// TwinCAT 3 PLC project PLCMotionOOP
// ProgramVersion: 3.1.4024.0
// libraries:
//   Tc2_MC2, * (Beckhoff Automation GmbH)
//   Tc2_Standard, * (Beckhoff Automation GmbH)
//   Tc2_System, * (Beckhoff Automation GmbH)
//   Tc3_Module, * (Beckhoff Automation GmbH)
// project tree:
//   MotionOOP/PLCOpenDefination/BeckhoffImplementation/ Axis.TcPOU
//   MotionOOP/PLCOpenDefination/Part1Definition/Enums/ AXIS_DIRECTION.TcDUT, AXIS_STATUS.TcDUT, MC_BUFFER_MODE.TcDUT, MC_COMBINE_MODE.TcDUT, MC_Direction.TcDUT, MC_Error.TcDUT, MC_ExecutionMode.TcDUT, MC_Source.TcDUT, MC_StartMode.TcDUT, MC_SYNC_MODE.TcDUT, MOTION_STATUS.TcDUT
//   MotionOOP/PLCOpenDefination/Part1Definition/GlobalConstants/ Constants.TcGVL
//   MotionOOP/PLCOpenDefination/Part1Definition/Interfaces/ itfAxis.TcIO, itfAxisCommand.TcIO, itfCamTable.TcIO, itfCommand.TcIO, itfContinuousAxisCommand.TcIO, itfSynchronizedAxisCommand.TcIO
//   MotionOOP/PLCOpenDefination/Part1Definition/Structs/ MC_CAM_REF.TcDUT, MC_COMMAND_REF.TcDUT
//   / PlcTask.TcTTO
//   POUs/ MAIN.TcPOU
// real-time tasks:
//   TASK PlcTask: cycle T#10ms, priority 20, ADS port 350
//   TASK PlcTask1: cycle T#10ms, priority 21, ADS port 351

CONFIGURATION PLCMotionOOP
    RESOURCE PLC ON TwinCAT3
        TASK PlcTask(INTERVAL := T#10ms, PRIORITY := 21);
        PROGRAM MAIN WITH PlcTask : MAIN;
    END_RESOURCE
END_CONFIGURATION

// ---- MotionOOP/PLCOpenDefination/Part1Definition/Enums/AXIS_DIRECTION.TcDUT
{attribute 'qualified_only' := ''}
{attribute 'strict' := ''}
TYPE AXIS_DIRECTION :
(
	DirectionPositive := 0,
	DirectionNegative := 1
);
END_TYPE

// ---- MotionOOP/PLCOpenDefination/Part1Definition/Enums/AXIS_STATUS.TcDUT
{attribute 'qualified_only' := ''}
{attribute 'strict' := ''}
TYPE AXIS_STATUS :
(
	ErrorStop := 0,
	Disabled := 1,
	Stopping := 2,
	Homing := 3,
	Standstill := 4,
	DiscreteMotion := 5,
	ContinuousMotion := 6,
	SynchronizedMotion := 7
);
END_TYPE

// ---- MotionOOP/PLCOpenDefination/Part1Definition/Enums/MC_BUFFER_MODE.TcDUT
{attribute 'qualified_only' := ''}
{attribute 'strict' := ''}
TYPE MC_BUFFER_MODE :
(
	mcAborting := 0,
	mcBuffered := 1,
	mcBlendingLow := 2,
	mcBlendingPrevious := 3,
	mcBlendingNext := 4,
	mcBlendingHigh := 5
);
END_TYPE

// ---- MotionOOP/PLCOpenDefination/Part1Definition/Enums/MC_COMBINE_MODE.TcDUT
{attribute 'qualified_only' := ''}
{attribute 'strict' := ''}
TYPE MC_COMBINE_MODE :
(
	enum_member := 0
);
END_TYPE

// ---- MotionOOP/PLCOpenDefination/Part1Definition/Enums/MC_Direction.TcDUT
{attribute 'qualified_only' := ''}
{attribute 'strict' := ''}
TYPE MC_Direction :
(
	mcPositiveDirection := 0,
	mcShortestWay := 1,
	mcNegativeDirection := 2,
	mcCurrentDirection := 3
);
END_TYPE

// ---- MotionOOP/PLCOpenDefination/Part1Definition/Enums/MC_Error.TcDUT
///{attribute 'conditionalshow' := 'SomeText'}
///{attribute 'conditionalshow'}
///{attribute 'hide'}
{attribute 'qualified_only' := ''}
TYPE MC_Error :
(
	NO_ERROR,
	TIME_OUT
);
END_TYPE

// ---- MotionOOP/PLCOpenDefination/Part1Definition/Enums/MC_ExecutionMode.TcDUT
{attribute 'qualified_only' := ''}
{attribute 'strict' := ''}
TYPE MC_ExecutionMode :
(
	mcImmediatly := 0,
	mcQueue := 1
);
END_TYPE

// ---- MotionOOP/PLCOpenDefination/Part1Definition/Enums/MC_Source.TcDUT
{attribute 'qualified_only' := ''}
{attribute 'strict' := ''}
TYPE MC_Source :
(
	mcSetValue := 0,
	mcActualValue := 1
);
END_TYPE

// ---- MotionOOP/PLCOpenDefination/Part1Definition/Enums/MC_StartMode.TcDUT
{attribute 'qualified_only' := ''}
{attribute 'strict' := ''}
TYPE MC_StartMode :
(
	mcAbsolute := 0,
	mcRelative := 1,
	mcRampIn := 2
);
END_TYPE

// ---- MotionOOP/PLCOpenDefination/Part1Definition/Enums/MC_SYNC_MODE.TcDUT
{attribute 'qualified_only' := ''}
{attribute 'strict' := ''}
TYPE MC_SYNC_MODE :
(
	enum_member := 0
);
END_TYPE

// ---- MotionOOP/PLCOpenDefination/Part1Definition/Enums/MOTION_STATUS.TcDUT
{attribute 'qualified_only' := ''}
{attribute 'strict' := ''}
TYPE MOTION_STATUS :
(
	ConstantVelocity := 0,
	Accelerating := 1,
	Decelerating := 2
);
END_TYPE

// ---- MotionOOP/PLCOpenDefination/Part1Definition/Structs/MC_CAM_REF.TcDUT
TYPE MC_CAM_REF :
STRUCT
END_STRUCT
END_TYPE

// ---- MotionOOP/PLCOpenDefination/Part1Definition/Structs/MC_COMMAND_REF.TcDUT
TYPE MC_COMMAND_REF :
STRUCT
	CommandId: INT;
END_STRUCT
END_TYPE

// ---- MotionOOP/PLCOpenDefination/Part1Definition/GlobalConstants/Constants.TcGVL
///{attribute 'conditionalshow' := 'SomeText'}
///{attribute 'conditionalshow'}
///{attribute 'hide'}
VAR_GLOBAL
END_VAR

// ---- MotionOOP/PLCOpenDefination/Part1Definition/Interfaces/itfAxis.TcIO
INTERFACE itfAxis

METHOD AccelerationProfile : itfCommand
VAR_INPUT
	TimeScale: REAL;
	AccelerationScale: REAL;
	Offset: REAL;
	BufferMode: MC_BUFFER_MODE;
END_VAR
END_METHOD

PROPERTY ActualPosition : REAL
GET
END_GET
END_PROPERTY

PROPERTY ActualTorque : REAL
GET
END_GET
END_PROPERTY

PROPERTY ActualVelocity : REAL
GET
END_GET
END_PROPERTY

PROPERTY AxisWarning : BOOL
GET
END_GET
END_PROPERTY

METHOD CamIn : itfSynchronizedAxisCommand
VAR_INPUT
	Master: itfAxis;
	MasterOffset: REAL;
	SlaveOffset: REAL;
	MasterScaling: REAL;
	SlaveScaling: REAL;
	MasterStartDistance: REAL;
	MasterSyncPosition: REAL;
	StartMode: MC_StartMode;
	MasterValueSource: MC_Source;
	CamTable: itfCamTable;
	BufferMode: MC_BUFFER_MODE;
END_VAR
END_METHOD

METHOD CombineAxes : itfSynchronizedAxisCommand
VAR_INPUT
	Master1: itfAxis;
	Master2: itfAxis;
	CombineMode: MC_COMBINE_MODE;
	GearRatioNumeratorM1: INT;
	GearRatioDenominatorM1: INT;
	GearRatioNumeratorM2: INT;
	GearRatioDenominatorM2: INT;
	MasterValueSourceM1: MC_SOURCE;
	MasterValueSourceM2: MC_SOURCE;
	BufferMode: MC_BUFFER_MODE;
END_VAR
END_METHOD

PROPERTY CommunicationReady : BOOL
GET
END_GET
END_PROPERTY

PROPERTY Direction : AXIS_DIRECTION
GET
END_GET
END_PROPERTY

PROPERTY ErrorId : WORD
GET
END_GET
END_PROPERTY

METHOD GearIn : itfSynchronizedAxisCommand
VAR_INPUT
	Master: itfAxis;
	Ratio: REAL;
	MasterValueSource: INT;
	Acceleration: REAL;
	Deceleration: REAL;
	Jerk: REAL;
	BufferMode: MC_BUFFER_MODE;
END_VAR
END_METHOD

METHOD GearInPos : itfSynchronizedAxisCommand
VAR_INPUT
	Master: itfAxis;
	RatioNumerator: REAL;
	RatioDenominator: REAL;
	MasterValueSource: MC_SOURCE;
	MasterSyncPosition: REAL;
	SlaveSyncPosition: REAL;
	SyncMode: MC_SYNC_MODE;
	MasterStartDistance: REAL;
	Velocity: REAL;
	Acceleration: REAL;
	Deceleration: REAL;
	Jerk: REAL;
	BufferMode: MC_BUFFER_MODE;
END_VAR
END_METHOD

METHOD Halt : itfAxisCommand
VAR_INPUT
	Deceleration: REAL;
	Jerk: REAL;
	BufferMode: MC_BUFFER_MODE;
END_VAR
END_METHOD

METHOD HaltSuperimposed : itfAxisCommand
VAR_INPUT
	Deceleration: REAL;
	Jerk: REAL;
END_VAR
END_METHOD

METHOD Home : itfAxisCommand
VAR_INPUT
	Position: REAL;
	Velocity: REAL;
	EndVelocity: REAL;
	Acceleration: REAL;
	Deceleration: REAL;
	Jerk: REAL;
	Direction: MC_Direction;
	HomingMode: INT;
	BufferMode: MC_BUFFER_MODE;
END_VAR
END_METHOD

PROPERTY HomeAbsSwitch : BOOL
GET
END_GET
END_PROPERTY

PROPERTY IsHomed : BOOL
GET
END_GET
END_PROPERTY

PROPERTY LimitSwitchNegative : BOOL
GET
END_GET
END_PROPERTY

PROPERTY LimitSwitchPositive : BOOL
GET
END_GET
END_PROPERTY

PROPERTY MotionStatus : MOTION_STATUS
GET
END_GET
END_PROPERTY

METHOD MoveAbsolute : itfAxisCommand
VAR_INPUT
	Position: REAL;
	Velocity: REAL;
	Acceleration: REAL;
	Deceleration: REAL;
	Jerk: REAL;
	Direction: MC_Direction;
	BufferMode: MC_BUFFER_MODE;
END_VAR
END_METHOD

METHOD MoveAdditive : itfAxisCommand
VAR_INPUT
	Distance: REAL;
	Velocity: REAL;
	Acceleration: REAL;
	Deceleration: REAL;
	Jerk: REAL;
	BufferMode: MC_BUFFER_MODE;
END_VAR
END_METHOD

METHOD MoveContinuousAbsolute : itfContinuousAxisCommand
VAR_INPUT
	Position: REAL;
	EndVelocity: REAL;
	Velocity: REAL;
	Acceleration: REAL;
	Deceleration: REAL;
	Jerk: REAL;
	Direction: MC_DIRECTION;
	BufferMode: MC_BUFFER_MODE;
END_VAR
END_METHOD

METHOD MoveContinuousRelative : itfContinuousAxisCommand
VAR_INPUT
	Distance: REAL;
	EndVelocity: REAL;
	Velocity: REAL;
	Acceleration: REAL;
	Deceleration: REAL;
	Jerk: REAL;
	Direction: MC_DIRECTION;
	BufferMode: MC_BUFFER_MODE;
END_VAR
END_METHOD

METHOD MoveRelative : itfAxisCommand
VAR_INPUT
	Distance: REAL;
	Velocity: REAL;
	Acceleration: REAL;
	Deceleration: REAL;
	Jerk: REAL;
	BufferMode: MC_BUFFER_MODE;
END_VAR
END_METHOD

METHOD MoveSuperimposed : itfAxisCommand
VAR_INPUT
	Distance: REAL;
	VelocityDiff: REAL;
	Acceleration: REAL;
	Deceleration: REAL;
	Jerk: REAL;
END_VAR
END_METHOD

METHOD MoveVelocity : itfContinuousAxisCommand
VAR_INPUT
	Velocity: REAL;
	Acceleration: REAL;
	Deceleration: REAL;
	Jerk: REAL;
	Direction: MC_Direction;
	BufferMode: MC_BUFFER_MODE;
END_VAR
END_METHOD

METHOD PhasingAbsolute : itfSynchronizedAxisCommand
VAR_INPUT
	Master: itfAxis;
	PhaseShift: REAL;
	Velocity: REAL;
	Acceleration: REAL;
	Deceleration: REAL;
	Jerk: REAL;
	BufferMode: MC_BUFFER_MODE;
END_VAR
END_METHOD

METHOD PhasingRelative : itfSynchronizedAxisCommand
VAR_INPUT
	Master: itfAxis;
	PhaseShift: REAL;
	Velocity: REAL;
	Acceleration: REAL;
	Deceleration: REAL;
	Jerk: REAL;
	BufferMode: MC_BUFFER_MODE;
END_VAR
END_METHOD

METHOD PositionProfile : itfCommand
VAR_INPUT
	TimeScale: REAL;
	PositionScale: REAL;
	Offset: REAL;
	BufferMode: MC_BUFFER_MODE;
END_VAR
END_METHOD

METHOD Power : itfCommand
VAR_INPUT
	Enable: BOOL;
	EnablePositive: BOOL;
	EnableNegative: BOOL;
END_VAR
END_METHOD

PROPERTY PowerOn : BOOL
GET
END_GET
END_PROPERTY

METHOD ReadBoolParameter : MC_Error
VAR_INPUT
	ParameterNumber: INT;
END_VAR
VAR_OUTPUT
	Value: BOOL;
END_VAR
END_METHOD

METHOD ReadParameter : MC_Error
VAR_INPUT
	ParameterNumber: INT;
END_VAR
VAR_OUTPUT
	Value: REAL;
END_VAR
END_METHOD

PROPERTY ReadyForPowerOn : BOOL
GET
END_GET
END_PROPERTY

METHOD Release : MC_Error
END_METHOD

METHOD Reset : itfCommand
END_METHOD

METHOD SetOverride : MC_Error
VAR_INPUT
	VelFactor: REAL;
	AccFactor: REAL;
	JerkFactor: REAL;
END_VAR
END_METHOD

METHOD SetPosition : itfCommand
VAR_INPUT
	Position: REAL;
	Relative: BOOL;
	ExecutionMode: MC_ExecutionMode;
END_VAR
END_METHOD

PROPERTY Simulation : BOOL
GET
END_GET
END_PROPERTY

PROPERTY Status : AXIS_STATUS
GET
END_GET
END_PROPERTY

METHOD Stop : itfAxisCommand
VAR_INPUT
	Deceleration: REAL;
	Jerk: REAL;
END_VAR
END_METHOD

METHOD TorqueControl : itfAxisCommand
VAR_INPUT
	Torque: REAL;
	TorqueRamp: REAL;
	Velocity: REAL;
	Acceleration: REAL;
	Deceleration: REAL;
	Jerk: REAL;
	Direction: MC_DIRECTION;
	BufferMode: MC_BUFFER_MODE;
END_VAR
END_METHOD

METHOD VelocityProfile : itfCommand
VAR_INPUT
	TimeScale: REAL;
	VelocityScale: REAL;
	Offset: REAL;
	BufferMode: MC_BUFFER_MODE;
END_VAR
END_METHOD

METHOD WriteBoolParameter : MC_Error
VAR_INPUT
	ParameterNumber: INT;
	Value: BOOL;
END_VAR
END_METHOD

METHOD WriteParameter : MC_Error
VAR_INPUT
	ParameterNumber: INT;
	Value: REAL;
END_VAR
END_METHOD

END_INTERFACE

// ---- MotionOOP/PLCOpenDefination/Part1Definition/Interfaces/itfAxisCommand.TcIO
INTERFACE itfAxisCommand EXTENDS itfCommand

METHOD Update : MC_Error
VAR_INPUT
	Position: REAL;
	Velocity: REAL;
	EndVelocity: REAL;
	Acceleration: REAL;
	Deceleration: REAL;
	Jerk: REAL;
END_VAR
END_METHOD

END_INTERFACE

// ---- MotionOOP/PLCOpenDefination/Part1Definition/Interfaces/itfCamTable.TcIO
INTERFACE itfCamTable

METHOD Select : itfCommand
VAR_INPUT
	Periodic: BOOL;
	MasterAbsolute: BOOL;
	SlaveAbsolute: BOOL;
	CamTable: MC_CAM_REF;
END_VAR
END_METHOD

END_INTERFACE

// ---- MotionOOP/PLCOpenDefination/Part1Definition/Interfaces/itfCommand.TcIO
INTERFACE itfCommand

METHOD Abort : MC_Error
END_METHOD

PROPERTY Active : BOOL
GET
END_GET
END_PROPERTY

PROPERTY Busy : BOOL
GET
END_GET
END_PROPERTY

PROPERTY Command : MC_COMMAND_REF
GET
END_GET
END_PROPERTY

PROPERTY CommandAborted : BOOL
GET
END_GET
END_PROPERTY

PROPERTY Done : BOOL
GET
END_GET
END_PROPERTY

PROPERTY Error : BOOL
GET
END_GET
END_PROPERTY

PROPERTY ErrorId : MC_Error
GET
END_GET
END_PROPERTY

METHOD Wait : MC_Error
VAR_INPUT
	Timeout: TIME;
	AbortOnTimeout: BOOL;
END_VAR
END_METHOD

END_INTERFACE

// ---- MotionOOP/PLCOpenDefination/Part1Definition/Interfaces/itfContinuousAxisCommand.TcIO
INTERFACE itfContinuousAxisCommand EXTENDS itfAxisCommand

PROPERTY InVelocity : BOOL
GET
END_GET
END_PROPERTY

END_INTERFACE

// ---- MotionOOP/PLCOpenDefination/Part1Definition/Interfaces/itfSynchronizedAxisCommand.TcIO
INTERFACE itfSynchronizedAxisCommand EXTENDS itfAxisCommand

PROPERTY InSync : BOOL
GET
END_GET
END_PROPERTY

END_INTERFACE

// ---- POUs/MAIN.TcPOU
PROGRAM MAIN
VAR
END_VAR

END_PROGRAM

// ---- MotionOOP/PLCOpenDefination/BeckhoffImplementation/Axis.TcPOU
FUNCTION_BLOCK Axis IMPLEMENTS itfAxis
VAR_INPUT
END_VAR
VAR_OUTPUT
END_VAR
VAR
END_VAR

{warning 'add method implementation '}
METHOD AccelerationProfile : itfCommand
VAR_INPUT
	TimeScale	: REAL;
	AccelerationScale	: REAL;
	Offset	: REAL;
	BufferMode	: MC_BUFFER_MODE;
END_VAR
END_METHOD

{warning 'add property implementation'}
PROPERTY ActualPosition : REAL
GET
END_GET
END_PROPERTY

{warning 'add property implementation'}
PROPERTY ActualTorque : REAL
GET
END_GET
END_PROPERTY

{warning 'add property implementation'}
PROPERTY ActualVelocity : REAL
GET
END_GET
END_PROPERTY

{warning 'add property implementation'}
PROPERTY AxisWarning : BOOL
GET
END_GET
END_PROPERTY

{warning 'add method implementation '}
METHOD CamIn : itfSynchronizedAxisCommand
VAR_INPUT
	Master	: itfAxis;
	MasterOffset	: REAL;
	SlaveOffset	: REAL;
	MasterScaling	: REAL;
	SlaveScaling	: REAL;
	MasterStartDistance	: REAL;
	MasterSyncPosition	: REAL;
	StartMode	: MC_StartMode;
	MasterValueSource	: MC_Source;
	CamTable	: itfCamTable;
	BufferMode	: MC_BUFFER_MODE;
END_VAR
END_METHOD

{warning 'add method implementation '}
METHOD CombineAxes : itfSynchronizedAxisCommand
VAR_INPUT
	Master1	: itfAxis;
	Master2	: itfAxis;
	CombineMode	: MC_COMBINE_MODE;
	GearRatioNumeratorM1	: INT;
	GearRatioDenominatorM1	: INT;
	GearRatioNumeratorM2	: INT;
	GearRatioDenominatorM2	: INT;
	MasterValueSourceM1	: MC_SOURCE;
	MasterValueSourceM2	: MC_SOURCE;
	BufferMode	: MC_BUFFER_MODE;
END_VAR
END_METHOD

{warning 'add property implementation'}
PROPERTY CommunicationReady : BOOL
GET
END_GET
END_PROPERTY

{warning 'add property implementation'}
PROPERTY Direction : AXIS_DIRECTION
GET
END_GET
END_PROPERTY

{warning 'add property implementation'}
PROPERTY ErrorId : WORD
GET
END_GET
END_PROPERTY

{warning 'add method implementation '}
METHOD GearIn : itfSynchronizedAxisCommand
VAR_INPUT
	Master	: itfAxis;
	Ratio	: REAL;
	MasterValueSource	: INT;
	Acceleration	: REAL;
	Deceleration	: REAL;
	Jerk	: REAL;
	BufferMode	: MC_BUFFER_MODE;
END_VAR
END_METHOD

{warning 'add method implementation '}
METHOD GearInPos : itfSynchronizedAxisCommand
VAR_INPUT
	Master	: itfAxis;
	RatioNumerator	: REAL;
	RatioDenominator	: REAL;
	MasterValueSource	: MC_SOURCE;
	MasterSyncPosition	: REAL;
	SlaveSyncPosition	: REAL;
	SyncMode	: MC_SYNC_MODE;
	MasterStartDistance	: REAL;
	Velocity	: REAL;
	Acceleration	: REAL;
	Deceleration	: REAL;
	Jerk	: REAL;
	BufferMode	: MC_BUFFER_MODE;
END_VAR
END_METHOD

{warning 'add method implementation '}
METHOD Halt : itfAxisCommand
VAR_INPUT
	Deceleration	: REAL;
	Jerk	: REAL;
	BufferMode	: MC_BUFFER_MODE;
END_VAR
END_METHOD

{warning 'add method implementation '}
METHOD HaltSuperimposed : itfAxisCommand
VAR_INPUT
	Deceleration	: REAL;
	Jerk	: REAL;
END_VAR
END_METHOD

{warning 'add method implementation '}
METHOD Home : itfAxisCommand
VAR_INPUT
	Position	: REAL;
	Velocity	: REAL;
	EndVelocity	: REAL;
	Acceleration	: REAL;
	Deceleration	: REAL;
	Jerk	: REAL;
	Direction	: MC_Direction;
	HomingMode	: INT;
	BufferMode	: MC_BUFFER_MODE;
END_VAR
END_METHOD

{warning 'add property implementation'}
PROPERTY HomeAbsSwitch : BOOL
GET
END_GET
END_PROPERTY

{warning 'add property implementation'}
PROPERTY IsHomed : BOOL
GET
END_GET
END_PROPERTY

{warning 'add property implementation'}
PROPERTY LimitSwitchNegative : BOOL
GET
END_GET
END_PROPERTY

{warning 'add property implementation'}
PROPERTY LimitSwitchPositive : BOOL
GET
END_GET
END_PROPERTY

{warning 'add property implementation'}
PROPERTY MotionStatus : MOTION_STATUS
GET
END_GET
END_PROPERTY

{warning 'add method implementation '}
METHOD MoveAbsolute : itfAxisCommand
VAR_INPUT
	Position	: REAL;
	Velocity	: REAL;
	Acceleration	: REAL;
	Deceleration	: REAL;
	Jerk	: REAL;
	Direction	: MC_Direction;
	BufferMode	: MC_BUFFER_MODE;
END_VAR
END_METHOD

{warning 'add method implementation '}
METHOD MoveAdditive : itfAxisCommand
VAR_INPUT
	Distance	: REAL;
	Velocity	: REAL;
	Acceleration	: REAL;
	Deceleration	: REAL;
	Jerk	: REAL;
	BufferMode	: MC_BUFFER_MODE;
END_VAR
END_METHOD

{warning 'add method implementation '}
METHOD MoveContinuousAbsolute : itfContinuousAxisCommand
VAR_INPUT
	Position	: REAL;
	EndVelocity	: REAL;
	Velocity	: REAL;
	Acceleration	: REAL;
	Deceleration	: REAL;
	Jerk	: REAL;
	Direction	: MC_DIRECTION;
	BufferMode	: MC_BUFFER_MODE;
END_VAR
END_METHOD

{warning 'add method implementation '}
METHOD MoveContinuousRelative : itfContinuousAxisCommand
VAR_INPUT
	Distance	: REAL;
	EndVelocity	: REAL;
	Velocity	: REAL;
	Acceleration	: REAL;
	Deceleration	: REAL;
	Jerk	: REAL;
	Direction	: MC_DIRECTION;
	BufferMode	: MC_BUFFER_MODE;
END_VAR
END_METHOD

{warning 'add method implementation '}
METHOD MoveRelative : itfAxisCommand
VAR_INPUT
	Distance	: REAL;
	Velocity	: REAL;
	Acceleration	: REAL;
	Deceleration	: REAL;
	Jerk	: REAL;
	BufferMode	: MC_BUFFER_MODE;
END_VAR
END_METHOD

{warning 'add method implementation '}
METHOD MoveSuperimposed : itfAxisCommand
VAR_INPUT
	Distance	: REAL;
	VelocityDiff	: REAL;
	Acceleration	: REAL;
	Deceleration	: REAL;
	Jerk	: REAL;
END_VAR
END_METHOD

{warning 'add method implementation '}
METHOD MoveVelocity : itfContinuousAxisCommand
VAR_INPUT
	Velocity	: REAL;
	Acceleration	: REAL;
	Deceleration	: REAL;
	Jerk	: REAL;
	Direction	: MC_Direction;
	BufferMode	: MC_BUFFER_MODE;
END_VAR
END_METHOD

{warning 'add method implementation '}
METHOD PhasingAbsolute : itfSynchronizedAxisCommand
VAR_INPUT
	Master	: itfAxis;
	PhaseShift	: REAL;
	Velocity	: REAL;
	Acceleration	: REAL;
	Deceleration	: REAL;
	Jerk	: REAL;
	BufferMode	: MC_BUFFER_MODE;
END_VAR
END_METHOD

{warning 'add method implementation '}
METHOD PhasingRelative : itfSynchronizedAxisCommand
VAR_INPUT
	Master	: itfAxis;
	PhaseShift	: REAL;
	Velocity	: REAL;
	Acceleration	: REAL;
	Deceleration	: REAL;
	Jerk	: REAL;
	BufferMode	: MC_BUFFER_MODE;
END_VAR
END_METHOD

{warning 'add method implementation '}
METHOD PositionProfile : itfCommand
VAR_INPUT
	TimeScale	: REAL;
	PositionScale	: REAL;
	Offset	: REAL;
	BufferMode	: MC_BUFFER_MODE;
END_VAR
END_METHOD

{warning 'add method implementation '}
METHOD Power : itfCommand
VAR_INPUT
	Enable	: BOOL;
	EnablePositive	: BOOL;
	EnableNegative	: BOOL;
END_VAR
END_METHOD

{warning 'add property implementation'}
PROPERTY PowerOn : BOOL
GET
END_GET
END_PROPERTY

{warning 'add method implementation '}
METHOD ReadBoolParameter : MC_Error
VAR_INPUT
	ParameterNumber	: INT;
END_VAR
VAR_OUTPUT
	Value	: BOOL;
END_VAR
END_METHOD

{warning 'add method implementation '}
METHOD ReadParameter : MC_Error
VAR_INPUT
	ParameterNumber	: INT;
END_VAR
VAR_OUTPUT
	Value	: REAL;
END_VAR
END_METHOD

{warning 'add property implementation'}
PROPERTY ReadyForPowerOn : BOOL
GET
END_GET
END_PROPERTY

{warning 'add method implementation '}
METHOD Release : MC_Error
END_METHOD

{warning 'add method implementation '}
METHOD Reset : itfCommand
END_METHOD

{warning 'add method implementation '}
METHOD SetOverride : MC_Error
VAR_INPUT
	VelFactor	: REAL;
	AccFactor	: REAL;
	JerkFactor	: REAL;
END_VAR
END_METHOD

{warning 'add method implementation '}
METHOD SetPosition : itfCommand
VAR_INPUT
	Position	: REAL;
	Relative	: BOOL;
	ExecutionMode	: MC_ExecutionMode;
END_VAR
END_METHOD

{warning 'add property implementation'}
PROPERTY Simulation : BOOL
GET
END_GET
END_PROPERTY

{warning 'add property implementation'}
PROPERTY Status : AXIS_STATUS
GET
END_GET
END_PROPERTY

{warning 'add method implementation '}
METHOD Stop : itfAxisCommand
VAR_INPUT
	Deceleration	: REAL;
	Jerk	: REAL;
END_VAR
END_METHOD

{warning 'add method implementation '}
METHOD TorqueControl : itfAxisCommand
VAR_INPUT
	Torque	: REAL;
	TorqueRamp	: REAL;
	Velocity	: REAL;
	Acceleration	: REAL;
	Deceleration	: REAL;
	Jerk	: REAL;
	Direction	: MC_DIRECTION;
	BufferMode	: MC_BUFFER_MODE;
END_VAR
END_METHOD

{warning 'add method implementation '}
METHOD VelocityProfile : itfCommand
VAR_INPUT
	TimeScale	: REAL;
	VelocityScale	: REAL;
	Offset	: REAL;
	BufferMode	: MC_BUFFER_MODE;
END_VAR
END_METHOD

{warning 'add method implementation '}
METHOD WriteBoolParameter : MC_Error
VAR_INPUT
	ParameterNumber	: INT;
	Value	: BOOL;
END_VAR
END_METHOD

{warning 'add method implementation '}
METHOD WriteParameter : MC_Error
VAR_INPUT
	ParameterNumber	: INT;
	Value	: REAL;
END_VAR
END_METHOD

END_FUNCTION_BLOCK
